FUNCTION_BLOCK FB_Timer
VAR_INPUT
	bStart          : BOOL := FALSE;
	bStop			: BOOL := FALSE;
END_VAR
VAR_OUTPUT
    tDifference     : TIME;
END_VAR
VAR
    StartTrigger,
	StopTrigger		: R_TRIG;
    StartTime    	: TIME;
    StopTime    	: TIME;
END_VAR

(*
Timer functionblock

Source:
https://infosys.beckhoff.de/index.php?content=../content/1031/tc3_plc_intro/2529365899.html&id=
*)
StartTrigger(CLK := bStart);
StopTrigger(CLK := bStop);

IF StartTrigger.Q THEN
    StartTime  := TIME();
END_IF

IF StopTrigger.Q THEN
    StopTime  := TIME();
    tDifference   := StopTime - StartTime;    // The difference will be T#5s
END_IF

END_FUNCTION_BLOCK

(* stored: Version 1.1.0.1, ProductVersion 3.1.4024.9
   POU FB_Timer: Id {51d55881-1840-43a3-abc1-8de5ef122133}, SpecialFunc None *)
